FUNCTION_BLOCK fb_motor_1
VAR_INPUT
	bStart, bStop : BOOL;
	
END_VAR
VAR_OUTPUT
	bStatus : BOOL;
END_VAR
VAR
END_VAR

END_FUNCTION_BLOCK

(* stored: Version 1.1.0.1, ProductVersion 3.1.4024.11
   POU fb_motor_1: Id {22f2864a-bac4-4277-8769-d0e239c058a6}, SpecialFunc None *)
